// TIA Portal V20 export
TYPE "LConSMC_typeTaperInput"
// stored: Access Published
   STRUCT
      enable : Bool := FALSE;   // TRUE: Funktionsbaustein aktivieren / TRUE: Enable function block
      taperMode : Int;   // Art der Kennlinie: 0: Keine Kennlinie 1: Lineare Kennlinie 2: Hyperbolische Kennlinie (maximale Reduktion am Zieldurchmesser) 3: Hyperbolische Kennlinie (Maximale Reduktion bei Unendlich) 4: Stützpunkttabelle / Tension taper characteristik 0: No taper 1: Linear taper characteristic 2: Hyperbolic taper characteristic (max. reduction at target diameter) 3: Hyperbolic taper characteristic (max. reduction at infinite diameter) 4: Breakpoint table
      diamActVal : LReal := 0.0;   // [ m oder inch ] Aktueller Durchmesser / [m or inch] Actual diameter value
      upperLimitTaper : LReal := 100.0;   // [%] Maximale Reduktion / [%] Maximum tension reduction
      lowerLimitTaper : LReal := 0.0;   // [%] Minimale Reduktion / [%] Minimum tension reduction
      taperRatio : LReal := 0.0;   // [%] Maximale Zugabsenkung bei "taperDiameterMax" (0-100%) Nur relevante für "taperMode" = 1-3 / [%] Maximum tension reduction at "taperDiameterMax" (0-100%) Only used if "taperMode" = 1-3
      taperDiameterStart : LReal := 0.2;   // [m oder inch] Startdurchmesser für die Reduktion / [m or inch] Diameter starting value for the tension reduction
      taperDiameterMax : LReal := 1.0;   // [m oder inch] maximaler Durchmesserwert. Wert am dem maximale Zugabsenkung gilt bei "taperMode" = 1 oder 2 / [m or inch] Maximum diameter value. Diameter at which the maximum tension reduction is active for "taperMode" = 1 or 2
      NoOfBreakpoints : Int := 20;   // Anzahl an verwendeten Stützpunkten (nur bei "taperMode" = 4) / Number of break points for breakpoint table if "taperMode" = 4
      tensionValues : "LConSMC_typeBreakPointTable";   // Stützpunkttabell für Zugabsenkungswerte im "taperMode" = 4 / Breakpoint table for tension reduction values if "taperMode" = 4
      diametervalues : "LConSMC_typeBreakPointTable";   // Stützpunkttabell für Durchmesserwerte im "taperMode" = 4 / Breakpoint table for diameter values if "taperMode" = 4
   END_STRUCT;
   // tensionValues.values[0..19] := 0.0;
   // diametervalues.values[0..19] := 0.0;
END_TYPE
